Universal Robots URScript: movep03.script

# movep:
# Set tcp: Use active tcp
# Tool speed : 250mm/s
# Tool acceleration : 1200mm/s2
# Blend with radius: 25mm
# waypoint1: feature view, xyz-RxRyRz (radian), Joint positions (degree)
# Use shared blend radius
# use shared parameters
# CircleMove: Fixed

def unnamed():
  global _hidden_verificationVariable=0
  step_count_ac8f1428_20c9_4a11_9ad0_dea55935d903 = 0.0
  thread Step_Counter_Thread_69af334b_b9fd_470e_a038_70c70d09c98e():
    while (True):
      step_count_ac8f1428_20c9_4a11_9ad0_dea55935d903 = step_count_ac8f1428_20c9_4a11_9ad0_dea55935d903 + 1.0
      sync()
    end
  end
  run Step_Counter_Thread_69af334b_b9fd_470e_a038_70c70d09c98e()
  set_target_payload(1.000000, [0.000000, 0.000000, 0.000000], [0.001539, 0.001539, 0.001539, 0.000000, 0.000000, 0.000000])
  set_tcp(p[0.0,0.0,0.0,0.0,0.0,0.0])
  set_tool_communication(False, 115200, 0, 1, 1.5, 3.5)
  set_tool_output_mode(0)
  set_tool_digital_output_mode(0, 1)
  set_tool_digital_output_mode(1, 1)
  set_tool_voltage(0)
  set_safety_mode_transition_hardness(1)
  set_standard_analog_input_domain(0, 1)
  set_standard_analog_input_domain(1, 1)
  set_tool_analog_input_domain(0, 1)
  set_tool_analog_input_domain(1, 1)
  set_analog_outputdomain(0, 0)
  set_analog_outputdomain(1, 0)
  set_input_actions_to_default()
  set_gravity([0.0, 0.0, 9.82])
  global Waypoint_1_p=p[-.136861537556, -.267180821738, .146971261118, -.001221359682, 3.116276528482, .038891915637]
  global Waypoint_1_q=[-1.6006999999999998, -1.7271, -2.2029999999999994, -0.8079999999999998, 1.5951, -0.030999999999999694]
  global ViaPoint_1_p=p[-.081219204219, -.230938488394, .146971261016, -.001221359682, 3.116276528481, .038891915639]
  global ViaPoint_1_q=[-1.3572936542112464, -1.4767886774316956, -2.469805077068303, -0.7848910134045077, 1.600579772274861, 0.2124344156522661]
  global EndPoint_1_p=p[-.036476870897, -.204296155036, .176013594340, .073926233660, 3.114816737594, .037931119442]
  global EndPoint_1_q=[-1.0834902626246494, -1.107083166129624, -2.5274140097160096, -1.0865766570825883, 1.6050920680674243, 0.5346156815996634]
  while (True):
    $ 1 "Robot Program"
    $ 2 "MoveP"
    $ 3 "Waypoint_1" "breakAfter"
    movep(Waypoint_1_p, a=1.2, v=0.25, r=0.025)
    $ 4 "CircleMove"
    $ 5 "ViaPoint_1" "noBreak"
    $ 6 "EndPoint_1" "breakAfter"
    movec(ViaPoint_1_p, EndPoint_1_p, a=1.2, v=0.25, r=0.025, mode=1)
  end
end
